FUNCTION_BLOCK E_SPLIT7
  (* Version 1.0, 2005-09-22, Goran Cengic, Chalmers *)
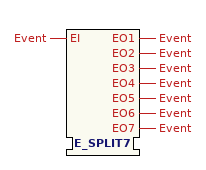
  EVENT_INPUT
    EI;
  END_EVENT
  EVENT_OUTPUT
    EO1;
    EO2;
    EO3;
    EO4;
    EO5;
    EO6;
    EO7;
  END_EVENT
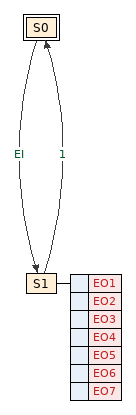
  EC_STATES
    S0;
    S1 : -> EO1, -> EO2, -> EO3, -> EO4, -> EO5, -> EO6, -> EO7;
  END_STATES
  EC_TRANSITIONS
    S0 TO S1 := EI;
    S1 TO S0 := 1;
  END_TRANSITIONS
END_FUNCTION_BLOCK
